// TIA Portal V18 export
// export: Created 2026-06-13T06:09:37.3076779Z, ExportSetting WithDefaults, DisplayName Totally Integrated Automation Portal, DisplayVersion V18, DisplayName TIA Portal Openness, DisplayVersion V18, DisplayName TIA Portal Version Control Interface, DisplayVersion V18, DisplayName STEP 7 Professional, DisplayVersion V18, DisplayName STEP 7 Safety, DisplayVersion V18, DisplayName WinCC Professional, DisplayVersion V18
ORGANIZATION_BLOCK "OB31_PID_PLC2_Bon4"   // OB31, LAD, CyclicInterrupt
{ S7_Optimized_Access := 'TRUE' }
VERSION : 0.1
// stored: AutoNumber true, IsIECCheckEnabled false, SetENOAutomatically false
   VAR_INPUT
      Initial_Call : Bool;   // Initial call of this OB
      Event_Count : Int;   // Events discarded
   END_VAR
BEGIN

REGION Network 1: Initialize PID Bon 4 Kp parameter
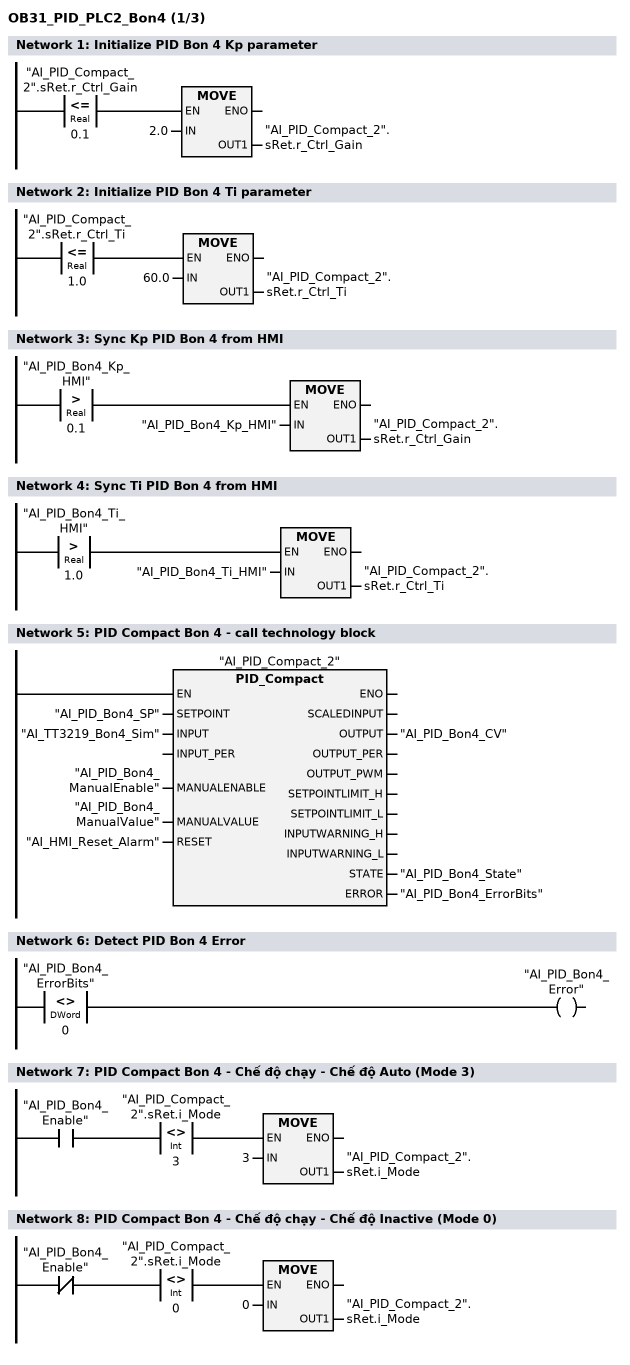
   RUNG wire#powerrail
      { S7_Templates := "SrcType := Real" } LE_Contact(in1 := "AI_PID_Compact_2".sRet.r_Ctrl_Gain, in2 := 0.1)
      { S7_GenerateENO := "TRUE" } Move(in := 2.0, out1 => "AI_PID_Compact_2".sRet.r_Ctrl_Gain)
   END_RUNG
   // the same network as SCL:
   IF "AI_PID_Compact_2".sRet.r_Ctrl_Gain <= 0.1 THEN "AI_PID_Compact_2".sRet.r_Ctrl_Gain := 2.0; END_IF;
END_REGION

REGION Network 2: Initialize PID Bon 4 Ti parameter
   RUNG wire#powerrail
      { S7_Templates := "SrcType := Real" } LE_Contact(in1 := "AI_PID_Compact_2".sRet.r_Ctrl_Ti, in2 := 1.0)
      { S7_GenerateENO := "TRUE" } Move(in := 60.0, out1 => "AI_PID_Compact_2".sRet.r_Ctrl_Ti)
   END_RUNG
   // the same network as SCL:
   IF "AI_PID_Compact_2".sRet.r_Ctrl_Ti <= 1.0 THEN "AI_PID_Compact_2".sRet.r_Ctrl_Ti := 60.0; END_IF;
END_REGION

REGION Network 3: Sync Kp PID Bon 4 from HMI
   RUNG wire#powerrail
      { S7_Templates := "SrcType := Real" } GT_Contact(in1 := "AI_PID_Bon4_Kp_HMI", in2 := 0.1)
      { S7_GenerateENO := "TRUE" } Move(in := "AI_PID_Bon4_Kp_HMI", out1 => "AI_PID_Compact_2".sRet.r_Ctrl_Gain)
   END_RUNG
   // the same network as SCL:
   IF "AI_PID_Bon4_Kp_HMI" > 0.1 THEN "AI_PID_Compact_2".sRet.r_Ctrl_Gain := "AI_PID_Bon4_Kp_HMI"; END_IF;
END_REGION

REGION Network 4: Sync Ti PID Bon 4 from HMI
   RUNG wire#powerrail
      { S7_Templates := "SrcType := Real" } GT_Contact(in1 := "AI_PID_Bon4_Ti_HMI", in2 := 1.0)
      { S7_GenerateENO := "TRUE" } Move(in := "AI_PID_Bon4_Ti_HMI", out1 => "AI_PID_Compact_2".sRet.r_Ctrl_Ti)
   END_RUNG
   // the same network as SCL:
   IF "AI_PID_Bon4_Ti_HMI" > 1.0 THEN "AI_PID_Compact_2".sRet.r_Ctrl_Ti := "AI_PID_Bon4_Ti_HMI"; END_IF;
END_REGION

REGION Network 5: PID Compact Bon 4 - call technology block
   RUNG wire#powerrail
      "AI_PID_Compact_2".PID_Compact(Setpoint := "AI_PID_Bon4_SP", Input := "AI_TT3219_Bon4_Sim", Input_PER :=, ManualEnable := "AI_PID_Bon4_ManualEnable", ManualValue := "AI_PID_Bon4_ManualValue", Reset := "AI_HMI_Reset_Alarm", ScaledInput =>, Output => "AI_PID_Bon4_CV", Output_PER =>, Output_PWM =>, SetpointLimit_H =>, SetpointLimit_L =>, InputWarning_H =>, InputWarning_L =>, State => "AI_PID_Bon4_State", Error => "AI_PID_Bon4_ErrorBits")
   END_RUNG
   // the same network as SCL:
   "AI_PID_Compact_2"(Setpoint := "AI_PID_Bon4_SP",   // PID_Compact
                      Input := "AI_TT3219_Bon4_Sim",
                      ManualEnable := "AI_PID_Bon4_ManualEnable",
                      ManualValue := "AI_PID_Bon4_ManualValue",
                      Reset := "AI_HMI_Reset_Alarm",
                      Output => "AI_PID_Bon4_CV",
                      State => "AI_PID_Bon4_State",
                      Error => "AI_PID_Bon4_ErrorBits");
END_REGION

REGION Network 6: Detect PID Bon 4 Error
   RUNG wire#powerrail
      { S7_Templates := "SrcType := DWord" } NE_Contact(in1 := "AI_PID_Bon4_ErrorBits", in2 := 0)
      Coil( "AI_PID_Bon4_Error" )
   END_RUNG
   // the same network as SCL:
   "AI_PID_Bon4_Error" := "AI_PID_Bon4_ErrorBits" <> 0;
END_REGION

REGION Network 7: PID Compact Bon 4 - Chế độ chạy - Chế độ Auto (Mode 3)
   RUNG wire#powerrail
      Contact( "AI_PID_Bon4_Enable" )
      { S7_Templates := "SrcType := Int" } NE_Contact(in1 := "AI_PID_Compact_2".sRet.i_Mode, in2 := 3)
      { S7_GenerateENO := "TRUE" } Move(in := 3, out1 => "AI_PID_Compact_2".sRet.i_Mode)
   END_RUNG
   // the same network as SCL:
   IF "AI_PID_Bon4_Enable" AND ("AI_PID_Compact_2".sRet.i_Mode <> 3) THEN
       "AI_PID_Compact_2".sRet.i_Mode := 3;
   END_IF;
END_REGION

REGION Network 8: PID Compact Bon 4 - Chế độ chạy - Chế độ Inactive (Mode 0)
   RUNG wire#powerrail
      I_Contact( "AI_PID_Bon4_Enable" )
      { S7_Templates := "SrcType := Int" } NE_Contact(in1 := "AI_PID_Compact_2".sRet.i_Mode, in2 := 0)
      { S7_GenerateENO := "TRUE" } Move(in := 0, out1 => "AI_PID_Compact_2".sRet.i_Mode)
   END_RUNG
   // the same network as SCL:
   IF NOT "AI_PID_Bon4_Enable" AND ("AI_PID_Compact_2".sRet.i_Mode <> 0) THEN
       "AI_PID_Compact_2".sRet.i_Mode := 0;
   END_IF;
END_REGION

REGION Network 9: Move PID Bon 4 CV to simulated heat valve
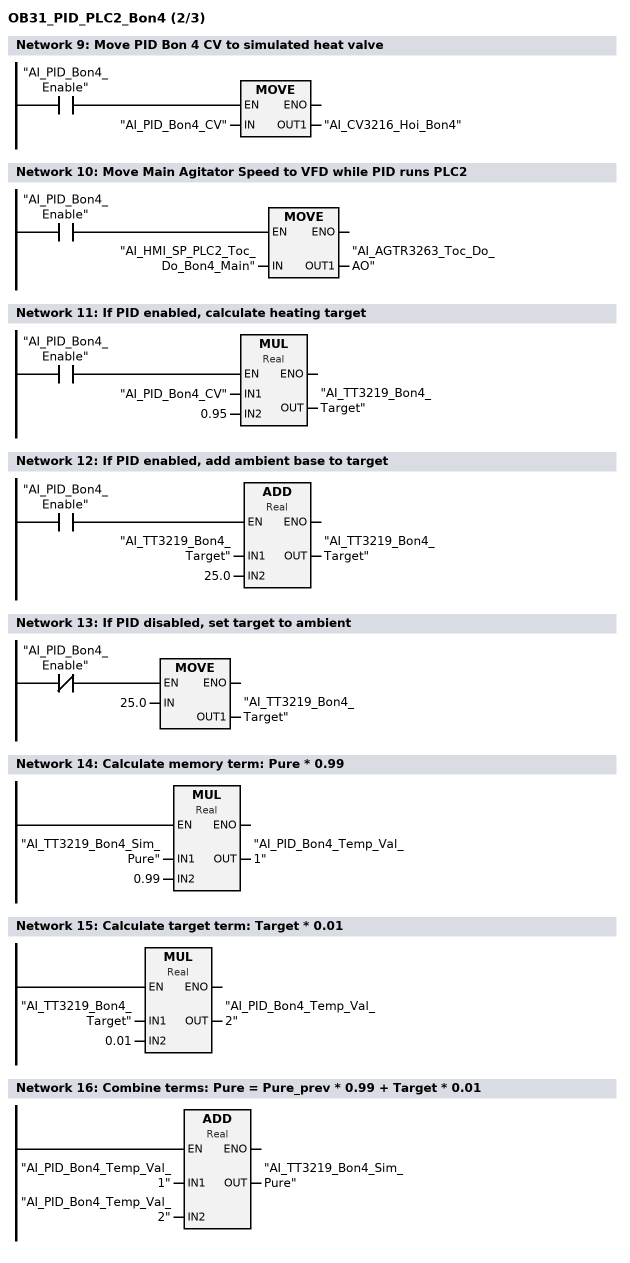
   RUNG wire#powerrail
      Contact( "AI_PID_Bon4_Enable" )
      { S7_GenerateENO := "TRUE" } Move(in := "AI_PID_Bon4_CV", out1 => "AI_CV3216_Hoi_Bon4")
   END_RUNG
   // the same network as SCL:
   IF "AI_PID_Bon4_Enable" THEN "AI_CV3216_Hoi_Bon4" := "AI_PID_Bon4_CV"; END_IF;
END_REGION

REGION Network 10: Move Main Agitator Speed to VFD while PID runs PLC2
   RUNG wire#powerrail
      Contact( "AI_PID_Bon4_Enable" )
      { S7_GenerateENO := "TRUE" } Move(in := "AI_HMI_SP_PLC2_Toc_Do_Bon4_Main", out1 => "AI_AGTR3263_Toc_Do_AO")
   END_RUNG
   // the same network as SCL:
   IF "AI_PID_Bon4_Enable" THEN "AI_AGTR3263_Toc_Do_AO" := "AI_HMI_SP_PLC2_Toc_Do_Bon4_Main"; END_IF;
END_REGION

REGION Network 11: If PID enabled, calculate heating target
   RUNG wire#powerrail
      Contact( "AI_PID_Bon4_Enable" )
      { S7_Templates := "SrcType := Real"; S7_GenerateENO := "TRUE" } Mul(in1 := "AI_PID_Bon4_CV", in2 := 0.95, out => "AI_TT3219_Bon4_Target")
   END_RUNG
   // the same network as SCL:
   IF "AI_PID_Bon4_Enable" THEN "AI_TT3219_Bon4_Target" := "AI_PID_Bon4_CV" * 0.95; END_IF;
END_REGION

REGION Network 12: If PID enabled, add ambient base to target
   RUNG wire#powerrail
      Contact( "AI_PID_Bon4_Enable" )
      { S7_Templates := "SrcType := Real"; S7_GenerateENO := "TRUE" } Add(in1 := "AI_TT3219_Bon4_Target", in2 := 25.0, out => "AI_TT3219_Bon4_Target")
   END_RUNG
   // the same network as SCL:
   IF "AI_PID_Bon4_Enable" THEN "AI_TT3219_Bon4_Target" := "AI_TT3219_Bon4_Target" + 25.0; END_IF;
END_REGION

REGION Network 13: If PID disabled, set target to ambient
   RUNG wire#powerrail
      I_Contact( "AI_PID_Bon4_Enable" )
      { S7_GenerateENO := "TRUE" } Move(in := 25.0, out1 => "AI_TT3219_Bon4_Target")
   END_RUNG
   // the same network as SCL:
   IF NOT "AI_PID_Bon4_Enable" THEN "AI_TT3219_Bon4_Target" := 25.0; END_IF;
END_REGION

REGION Network 14: Calculate memory term: Pure * 0.99
   RUNG wire#powerrail
      { S7_Templates := "SrcType := Real"; S7_GenerateENO := "TRUE" } Mul(in1 := "AI_TT3219_Bon4_Sim_Pure", in2 := 0.99, out => "AI_PID_Bon4_Temp_Val_1")
   END_RUNG
   // the same network as SCL:
   "AI_PID_Bon4_Temp_Val_1" := "AI_TT3219_Bon4_Sim_Pure" * 0.99;
END_REGION

REGION Network 15: Calculate target term: Target * 0.01
   RUNG wire#powerrail
      { S7_Templates := "SrcType := Real"; S7_GenerateENO := "TRUE" } Mul(in1 := "AI_TT3219_Bon4_Target", in2 := 0.01, out => "AI_PID_Bon4_Temp_Val_2")
   END_RUNG
   // the same network as SCL:
   "AI_PID_Bon4_Temp_Val_2" := "AI_TT3219_Bon4_Target" * 0.01;
END_REGION

REGION Network 16: Combine terms: Pure = Pure_prev * 0.99 + Target * 0.01
   RUNG wire#powerrail
      { S7_Templates := "SrcType := Real"; S7_GenerateENO := "TRUE" } Add(in1 := "AI_PID_Bon4_Temp_Val_1", in2 := "AI_PID_Bon4_Temp_Val_2", out => "AI_TT3219_Bon4_Sim_Pure")
   END_RUNG
   // the same network as SCL:
   "AI_TT3219_Bon4_Sim_Pure" := "AI_PID_Bon4_Temp_Val_1" + "AI_PID_Bon4_Temp_Val_2";
END_REGION

REGION Network 17: Increment simulation counter
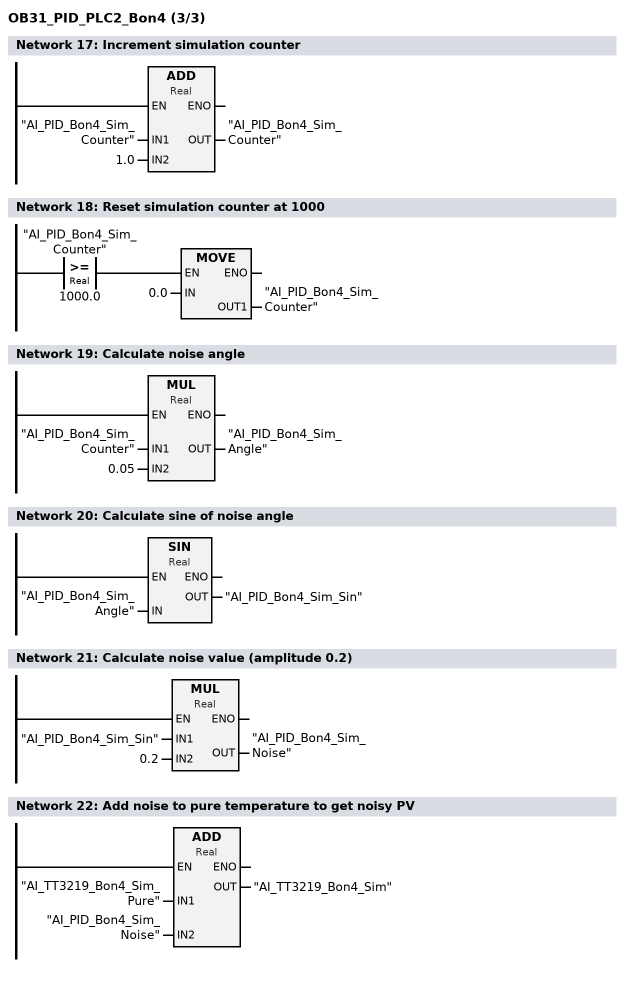
   RUNG wire#powerrail
      { S7_Templates := "SrcType := Real"; S7_GenerateENO := "TRUE" } Add(in1 := "AI_PID_Bon4_Sim_Counter", in2 := 1.0, out => "AI_PID_Bon4_Sim_Counter")
   END_RUNG
   // the same network as SCL:
   "AI_PID_Bon4_Sim_Counter" := "AI_PID_Bon4_Sim_Counter" + 1.0;
END_REGION

REGION Network 18: Reset simulation counter at 1000
   RUNG wire#powerrail
      { S7_Templates := "SrcType := Real" } GE_Contact(in1 := "AI_PID_Bon4_Sim_Counter", in2 := 1000.0)
      { S7_GenerateENO := "TRUE" } Move(in := 0.0, out1 => "AI_PID_Bon4_Sim_Counter")
   END_RUNG
   // the same network as SCL:
   IF "AI_PID_Bon4_Sim_Counter" >= 1000.0 THEN "AI_PID_Bon4_Sim_Counter" := 0.0; END_IF;
END_REGION

REGION Network 19: Calculate noise angle
   RUNG wire#powerrail
      { S7_Templates := "SrcType := Real"; S7_GenerateENO := "TRUE" } Mul(in1 := "AI_PID_Bon4_Sim_Counter", in2 := 0.05, out => "AI_PID_Bon4_Sim_Angle")
   END_RUNG
   // the same network as SCL:
   "AI_PID_Bon4_Sim_Angle" := "AI_PID_Bon4_Sim_Counter" * 0.05;
END_REGION

REGION Network 20: Calculate sine of noise angle
   "AI_PID_Bon4_Sim_Sin" := SIN("AI_PID_Bon4_Sim_Angle");
END_REGION

REGION Network 21: Calculate noise value (amplitude 0.2)
   RUNG wire#powerrail
      { S7_Templates := "SrcType := Real"; S7_GenerateENO := "TRUE" } Mul(in1 := "AI_PID_Bon4_Sim_Sin", in2 := 0.2, out => "AI_PID_Bon4_Sim_Noise")
   END_RUNG
   // the same network as SCL:
   "AI_PID_Bon4_Sim_Noise" := "AI_PID_Bon4_Sim_Sin" * 0.2;
END_REGION

REGION Network 22: Add noise to pure temperature to get noisy PV
   RUNG wire#powerrail
      { S7_Templates := "SrcType := Real"; S7_GenerateENO := "TRUE" } Add(in1 := "AI_TT3219_Bon4_Sim_Pure", in2 := "AI_PID_Bon4_Sim_Noise", out => "AI_TT3219_Bon4_Sim")
   END_RUNG
   // the same network as SCL:
   "AI_TT3219_Bon4_Sim" := "AI_TT3219_Bon4_Sim_Pure" + "AI_PID_Bon4_Sim_Noise";
END_REGION
END_ORGANIZATION_BLOCK
